// TIA Portal project "Project" (V15.1)

(* hardware
DEVICE "S71500/ET200MP station_1"  S7-1500 station
   slot 0: "Rail_0"  Rack  6ES7 590-1***0-0AA0
   slot 1: "R00.m01.CPU"  CPU 1515F-2 PN  6ES7 515-2FM01-0AB0  V2.6
      slot 3: "CPU display_1"  6ES7591-1BA00-0AA0
   slot 2: "R00.m02.DI16x32HF"  DI 16x24VDC HF  6ES7 521-1BH00-0AB0  V2.2
   slot 3: "R00.m03.DQ16x24HF"  DQ 16x24VDC/0.5A HF  6ES7 522-1BH01-0AB0  V1.1
DEVICE "SINAMICS S_1"  AcxSinamics.Device.2x.S210
   slot 0: "Unit1.a01.Sync.Master"  S210 PN  6SL3210-5HB10-1xFx  V5.2
      slot 1: "PROFINET interface"  PROFINET
      slot 3: " Ethernet commissioning interface"  LAN
   slot 0: "Drive control"  S210 PN
      slot 200: "Power Module_1"  Drive control  6SL3210-5HB10-1xFx
      slot 1000: "Motor_1"  Drive control  1FK2xxx-xxxxx-xxxx
DEVICE "SINAMICS S_2"  AcxSinamics.Device.2x.S210
   slot 0: "Unit1.a02.Sync.Slave"  S210 PN  6SL3210-5HB10-1xFx  V5.2
      slot 1: "PROFINET interface"  PROFINET
      slot 3: " Ethernet commissioning interface"  LAN
   slot 0: "Drive control"  S210 PN
      slot 200: "Power Module_1"  Drive control  6SL3210-5HB10-1xFx
      slot 1000: "Motor_1"  Drive control  1FK2xxx-xxxxx-xxxx
DEVICE "R00.m99.HMI"  TP900 Comfort
   slot 0: "R00.m99.HMI"  TP900 Comfort  6AV2 124-0JC01-0AX0  15.1.0.0
   slot 1: "HMI_RT_1"  TP900 Comfort  6AV2 124-0JC01-0AX0  15.1.0.0
   slot 5: "R00.m99.HMI.IE_CP_1"  PROFINET Interface  15.0.1.0
      slot 1: "PROFINET Interface_1"  PROFINET Interface
         slot 1: "Port_1"  Port
         slot 2: "Port_2"  Port
   slot 7: "R00.m99.HMI.MPI/DP_CP_1"  MPI/DP Interface  15.0.1.0
*)

// ===== PLC "R00.m01.CPU"  CPU 1515F-2 PN =====

VAR_GLOBAL   // PLC tag table "Default tag table"
   "Unit1.a02_Actor_Interface_AddressIn" AT %I276.0 : "PD_TEL105_IN";
   "Unit1.a02_Actor_Interface_AddressOut" AT %Q276.0 : "PD_TEL105_OUT";
   "Unit1.a01_Actor_Interface_AddressIn" AT %I256.0 : "PD_TEL105_IN";
   "Unit1.a01_Actor_Interface_AddressOut" AT %Q256.0 : "PD_TEL105_OUT";
   "R00.m02.Ch0.ESTOP" AT %I0.0 : Bool;
   "R00.m02.Ch1.Reset" AT %I0.1 : Bool;
END_VAR

DATA_BLOCK "Main_Safety_RTG1_DB"   // DB1, F_DB
{ S7_Optimized_Access := 'TRUE' }
NAME : FUSI
VERSION : 0.1
// stored: InstanceOfName Main_Safety_RTG1
"Main_Safety_RTG1"
BEGIN
END_DATA_BLOCK

DATA_BLOCK "Unit1.a02"   // DB2, Motion_DB
{ S7_Optimized_Access := 'TRUE' }
AUTHOR : SIMATIC
FAMILY : MC_1500
VERSION : 4.0
// stored: InstanceOfName TO_PositioningAxis
"TO_PositioningAxis"
BEGIN
END_DATA_BLOCK

DATA_BLOCK "Unit1.a01"   // DB3, Motion_DB
{ S7_Optimized_Access := 'TRUE' }
AUTHOR : SIMATIC
FAMILY : MC_1500
VERSION : 4.0
// stored: InstanceOfName TO_SynchronousAxis
"TO_SynchronousAxis"
BEGIN
END_DATA_BLOCK

FUNCTION_BLOCK "Main_Safety_RTG1"   // FB1, F_FBD
{ S7_Optimized_Access := 'TRUE' }
VERSION : 0.1
BEGIN
END_FUNCTION_BLOCK

ORGANIZATION_BLOCK "Main"   // OB1, LAD, ProgramCycle
TITLE = "Main Program Sweep (Cycle)"
{ S7_Optimized_Access := 'TRUE' }
VERSION : 0.1
   VAR_INPUT
      Initial_Call : Bool;   // Initial call of this OB
      Remanence : Bool;   // =True, if remanent data are available
   END_VAR
BEGIN
END_ORGANIZATION_BLOCK

(* ===== HMI "HMI_RT_1" =====
system functions are stored by id; their names below are inferred from use
connection "HMI_Connection_1": ETHERNET, S7_1500_OMS

HMI tags "Default tag table"
   "Tag_ScreenNumber" : UInt, internal

screen "Root screen" 800x420, template "Template_1"
   on GenerateScreen: SetTag("Tag_ScreenNumber", 1)
   TextField "HmiScreenItemData" at 80,167 size 640x22; Text 'Welcome to R00.m99.HMI (TP900 Comfort)!'

Template "Template_1" 800x420
   Button "Exit" at 720,360 size 78x58; TextOff 'Exit'; PictureOff "ExitRuntime_TP900_Comfort_TR"; PictureOn "ExitRuntime_TP900_Comfort_TR"
      on Release: StopRuntime(0)
   Button "Template_Button" at 640,360 size 78x58; TextOff 'Text'
   Button "Template_Button_1" at 560,360 size 78x58; TextOff 'Text'
   Button "Template_Button_2" at 480,360 size 78x58; TextOff 'Text'
   Button "Template_Button_3" at 400,360 size 78x58; TextOff 'Text'
   Button "Template_Button_4" at 321,360 size 78x58; TextOff 'Text'
   Button "Template_Button_5" at 241,360 size 78x58; TextOff 'Text'
   Button "Template_Button_6" at 161,360 size 78x58; TextOff 'Text'
   Button "Template_Button_7" at 81,360 size 78x58; TextOff 'Text'
   Button "Start screen" at 1,360 size 78x58; TextOff 'Start screen'; PictureOff "NavigateHome_TP900_Comfort_TR"; PictureOn "NavigateHome_TP900_Comfort_TR"
      on Release: ActivateScreen("Root screen", 0)
*)